PROGRAM CraneSimulation
VAR
	fCyclicTime : LREAL := 0.01;
	
	fbCraneStatus : FB_CraneStatus;
	fbCraneMode : FB_CraneMode;
END_VAR

// Crane status state machine
fbCraneStatus(	bPower := Inputs.bOnSelector,
		 		bStart := Inputs.bStartButton, 
				bStop := Inputs.bStopButton, 
				bRunning := Parameters.stStateVariables.bRunning, 
				bError := Parameters.stStateVariables.bError,
				eCraneStatus => Outputs.eCraneStatus);

// Crane mode state machine
IF Parameters.stStateVariables.bRunning THEN
	fbCraneMode( 	bRunning := Parameters.stStateVariables.bRunning,
					bMode := Inputs.bAutoSelector,
					eCraneMode => Outputs.eCraneMode);
END_IF
	
// Calculate boom angle for visualization of simulation		
HMI.fBoomAngle := F_BoomAngle(	fCylinderX := HMI.fCylinderPositonReference);

// Simulation timer			
IF Parameters.stStateVariables.bRunning THEN
	Parameters.stStateVariables.fTime := Parameters.stStateVariables.fTime + fCyclicTime;
ELSE
	Parameters.stStateVariables.fTime := 0.0;
END_IF

END_PROGRAM

(* stored: Version 1.1.0.1, ProductVersion 3.1.4024.10
   POU CraneSimulation: Id {9db64730-0769-4523-9dc9-b42b5865fac6}, SpecialFunc None *)
